FUNCTION_BLOCK L2_L1Comm (* Basic Function Block Type *)
  (* Standard: 61499-2 *)
  (* Version 0.0, 2015-02-25, EQUEROL, UJI *)
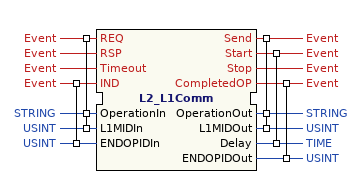
  EVENT_INPUT
    REQ WITH OperationIn, L1MIDIn; (* Send new operation request *)
    RSP; (* Operation reception confirmation *)
    Timeout; (* Communication timeout *)
    IND WITH ENDOPIDIn; (* Completed OP indication *)
  END_EVENT
  EVENT_OUTPUT
    Send WITH OperationOut, L1MIDOut; (* Send operation to Layer 1 *)
    Start WITH Delay; (* Start communication timeout *)
    Stop; (* Stop communication timeout *)
    CompletedOP WITH ENDOPIDOut; (* Completed Operation event *)
  END_EVENT
  VAR_INPUT
    OperationIn : STRING; (* String containing the serialized operation *)
    L1MIDIn : USINT; (* Layer 1 multicsat ID *)
    ENDOPIDIn : USINT; (* Operation end code *)
  END_VAR
  VAR_OUTPUT
    OperationOut : STRING; (* String containing the serialized operation *)
    L1MIDOut : USINT; (* Layer 1 multicast ID *)
    Delay : TIME; (* Timeout delay *)
    ENDOPIDOut : USINT; (* operation end code *)
  END_VAR
  VAR
    TOCounter : USINT := 0; (* Timeout counter *)
  END_VAR
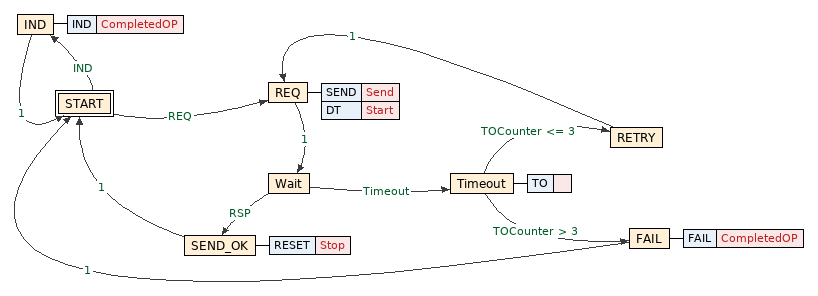
  EC_STATES
    START; (* Initial State *)
    REQ : SEND -> Send, DT -> Start; (* Normal execution *)
    Wait;
    SEND_OK : RESET -> Stop;
    Timeout : TO;
    RETRY;
    FAIL : FAIL -> CompletedOP;
    IND : IND -> CompletedOP;
  END_STATES
  EC_TRANSITIONS
    START TO REQ := REQ;
    REQ TO Wait := 1;
    Wait TO SEND_OK := RSP;
    SEND_OK TO START := 1;
    Wait TO Timeout := Timeout;
    Timeout TO FAIL := TOCounter > 3;
    Timeout TO RETRY := TOCounter <= 3;
    RETRY TO REQ := 1;
    FAIL TO START := 1;
    START TO IND := IND;
    IND TO START := 1;
  END_TRANSITIONS
  ALGORITHM SEND IN ST: (* Normally executed algorithm *)
OperationOut := OperationIn;
L1MIDOut := L1MIDIn;
  END_ALGORITHM
  ALGORITHM DT IN ST: (* Algo to parametrize the timeout *)
Delay := TIME#1500ms;
  END_ALGORITHM
  ALGORITHM RESET IN ST: (* Reset timeout counter *)
TOCounter := 0;
  END_ALGORITHM
  ALGORITHM TO IN ST: (* Communication timeout algo *)
TOCounter := TOCounter + 1;
  END_ALGORITHM
  ALGORITHM FAIL IN ST: (* Communication with L1 failure algo *)
TOCounter := 0;
(*Mark operation as failed but repeatable*)
ENDOPIDOut := 1;
  END_ALGORITHM
  ALGORITHM IND IN ST: (* Completed OP algo *)
ENDOPIDOut := ENDOPIDIn;
  END_ALGORITHM
END_FUNCTION_BLOCK
